TYPE "FeedMachine_CIn"
VERSION : 0.1
// Block: FeedMachine_CIn
   STRUCT
      Manager : FeedMachine_Manager;
      Bwd_ExtEnable : Bool;
      Fwd_ExtEnable : Bool;
      EnableManChangeVel : Bool;
      ExternalAlarms : Bool;
      VelocityOverride : Struct
         Enable : Bool;
         Value : LReal;
      END_STRUCT;
   END_STRUCT;

END_TYPE
